// TIA Portal V19 export
TYPE "LubrValve_Config"
// stored: Access Published
   STRUCT
      WorkMode : Int;   // 0:Work By CycleFdbk, 1:Work By Time, 2=Count Valve Cmd
      CounterMode : Int;   // 0:SpaceCounter, 1:OpCounter
      ValveType : Int;   // 0:Valve always ON, 1:Valve ON-OFF
      ManualCmdTimeOut : Time := T#5M;   // Time Out manual command
   END_STRUCT;
END_TYPE
